FUNCTION_BLOCK FB_ModuleBase EXTENDS FB_Component
VAR_INPUT
END_VAR
VAR_OUTPUT
END_VAR
VAR
	fbMembers:					FB_ListComponent;
	fbLoggerFactory:			FB_LoggerFactory;;
	fbTcLogger:					FB_TcLogger;
END_VAR

// https://github.com/PeterZerlauth/Tc3_Component

METHOD PROTECTED M_Aborted
VAR_INPUT
END_VAR
SUPER^.M_Aborted();
fbEvent.M_AddSTRING(P_Identifier);
fbEvent.M_Information('Module %s aborted, reset', '');
END_METHOD

METHOD PUBLIC M_Attach
VAR_INPUT
	Component:		I_Component;
END_VAR
Component.P_Event.P_Logger:= fbLoggerFactory;
fbMembers.M_Add(Component);
Component.P_Observer.M_Attach(THIS^);
fbObserver.M_Attach(Component);
END_METHOD

METHOD PUBLIC M_Cycle
VAR_INPUT
END_VAR
fbLoggerFactory();

SUPER^.M_Cycle();
END_METHOD

METHOD PUBLIC M_Dettach
VAR_INPUT
	Component:		I_Component;
END_VAR
Component.P_Event.P_Logger:= 0;
fbMembers.M_Remove(Component);
Component.P_Observer.M_Detach(THIS^);
fbObserver.M_Detach(Component);
END_METHOD

METHOD PROTECTED M_Idle
VAR_INPUT
END_VAR
SUPER^.M_Idle();
fbEvent.M_AddSTRING(P_Identifier);
fbEvent.M_Information('Module %s not started', '');
END_METHOD

METHOD PROTECTED M_Initialise
VAR_INPUT
END_VAR
SUPER^.M_Initialise();
fbEvent.P_Logger:= fbLoggerFactory;
fbLoggerFactory.M_Attach(fbTcLogger);
END_METHOD

METHOD Protected M_OnMode
VAR_INPUT
	eMode:							E_Mode;						// Current mode
	eModePrevious:					E_Mode;						// Previous mode	
END_VAR
CASE eMode OF
	E_Mode.Semiauto, E_Mode.Automatic:
		IF eModePrevious = E_Mode.Manual THEN
			fbEvent.M_AddSTRING(P_Identifier);
			fbEvent.M_Abort('Module %s was in manual mode', '');
		END_IF
END_CASE
END_METHOD

METHOD PROTECTED M_Resetting : BOOL
VAR_INPUT
END_VAR
M_Resetting:= SUPER^.M_Resetting();
fbMembers.M_Request(E_Request.Reset);
fbLoggerFactory.M_Reset();
END_METHOD

METHOD PROTECTED M_Resuming : BOOL // Return state complete
VAR_INPUT
END_VAR
M_Resuming:= fbMembers.M_Request(E_Request.Start);
END_METHOD

METHOD PROTECTED M_Running
VAR_INPUT
END_VAR
END_METHOD

METHOD PROTECTED M_Starting : BOOL
VAR_INPUT
END_VAR
M_Starting:= fbMembers.M_Request(E_Request.Start);
END_METHOD

METHOD PROTECTED M_Stopped
VAR_INPUT
END_VAR
SUPER^.M_Stopped();
fbEvent.M_AddSTRING(P_Identifier);
fbEvent.M_Information('Module %s stopped, reset', '');
END_METHOD

METHOD PROTECTED M_Unholding : BOOL // Return state complete
VAR_INPUT
END_VAR
M_Unholding:= fbMembers.M_Request(E_Request.Start);
END_METHOD

END_FUNCTION_BLOCK

(* stored: Version 1.1.0.1
   POU FB_ModuleBase: Id {0d3fc497-598e-0d21-1617-ce19be6391a0}, SpecialFunc None
   Method M_Aborted: Id {0b832f7f-4585-09d1-3d1d-4466841374ad}
   Method M_Attach: Id {579d130b-ed70-0843-1869-7cfcfab74d3d}
   Method M_Cycle: Id {ba6e3712-faea-4bef-b491-24a585067e68}
   Method M_Dettach: Id {a667402b-5023-09c1-34b6-30ca3f961f61}
   Method M_Idle: Id {6e9b6a1a-c168-0e2f-3b3d-1c86715a124a}
   Method M_Initialise: Id {d2ecc479-1ed6-0218-1db6-cf2c288ac295}
   Method M_OnMode: Id {8aa684a1-26e4-029d-2fa8-0e0341c2e439}
   Method M_Resetting: Id {61e3d89a-8bee-473b-9814-ba7482888f16}
   Method M_Resuming: Id {d9ef3688-d135-0f0b-1ce4-980e688e3f9f}
   Method M_Running: Id {8879f60a-43a4-0568-363b-e25a42eddf0c}
   Method M_Starting: Id {5a9fb78b-3ed4-0195-387d-72e3c96a0cbd}
   Method M_Stopped: Id {43b02a69-b318-0eb0-3e6f-2d210026cf6d}
   Method M_Unholding: Id {e6d01443-ae5b-0242-3775-c5c307506d4e} *)
